// TIA Portal V16 export
// export: Created 2021-05-28T04:18:29.314913Z, ExportSetting WithDefaults, DisplayName Totally Integrated Automation Portal, DisplayVersion V16 Update 4, DisplayName TIA Portal Version Control Interface, DisplayVersion V16 Update 2, DisplayName TIA Portal Openness, DisplayVersion V16 Update 4, DisplayName STEP 7 Professional, DisplayVersion V16 Update 4, DisplayName STEP 7 Safety, DisplayVersion V16, DisplayName WinCC Advanced, DisplayVersion V16 Update 4
FUNCTION_BLOCK "Main_Safety_RTG1"   // FB1, F_FBD
{ S7_Optimized_Access := 'TRUE' }
VERSION : 0.1
// stored: AutoNumber false, IsIECCheckEnabled false, UDAEnableTagReadback false
   VAR
      a_and_b : Bool;
      a_or_b : Bool;
      p_trig_state : Bool;
   END_VAR
   VAR_TEMP
      rising_a_or_b : Bool;
   END_VAR
   VAR_TEMP   // added for the SCL form of the ladder/FBD networks
      _w1 : Bool;
   END_VAR
BEGIN

REGION Network 1
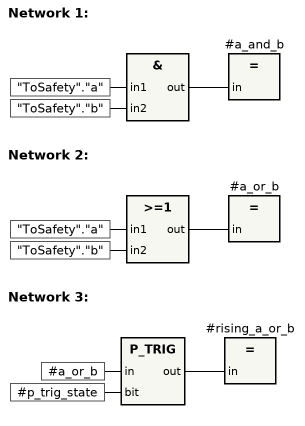
   #a_and_b := "ToSafety"."a" AND "ToSafety"."b";
END_REGION

REGION Network 2
   #a_or_b := "ToSafety"."a" OR "ToSafety"."b";
END_REGION

REGION Network 3
   #_w1 := #a_or_b AND NOT #p_trig_state;   // rising edge
   #p_trig_state := #a_or_b;
   #rising_a_or_b := #_w1;
END_REGION
END_FUNCTION_BLOCK
